FUNCTION FIELDBUS_PERCENT_TO_WORD
  (* Standard: SAE J1939; ISO 11783; Description: Copyright (c) 2023 HR Agrartechnik GmbH This program and the accompanying materials are made available under the terms of the Eclipse Public License 2.0 which is available at https://www.eclipse.org/legal/epl-2.0/ SPDX-License-Identifier: EPL-2.0 *)
  (* Version 1.0, 2023-10-21, franz *)
  PACKAGE signalprocessing;
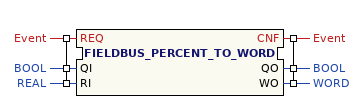
  EVENT_INPUT
    REQ WITH QI, RI;
  END_EVENT
  EVENT_OUTPUT
    CNF WITH QO, WO;
  END_EVENT
  VAR_INPUT
    QI : BOOL;
    RI : REAL;
  END_VAR
  VAR_OUTPUT
    QO : BOOL;
    WO : WORD;
  END_VAR
  BODY IN ST:
PACKAGE signalprocessing;

FUNCTION FIELDBUS_PERCENT_TO_WORD
VAR_INPUT
	QI : BOOL;
	RI : REAL;
END_VAR

VAR_OUTPUT
	QO : BOOL;
	WO : WORD;
END_VAR

QO := QI;
IF (TRUE = QI) THEN
	WO := UDINT_TO_WORD(REAL_TO_UDINT(RI * UDINT_TO_REAL(WORD_TO_UDINT(FIELDBUS_VALID_SIGNAL_W))));
END_IF;
END_FUNCTION
  END_BODY
END_FUNCTION
